PROGRAM MAIN
VAR
	//Matrix instances
	fbDispenseMatrix : FB_Matrix;
	fbInletMatrix : FB_Matrix;
	fbFillMatrix : FB_Matrix;

	//Instance of fbIO for IO updates
	fbIO : FB_IO;
	
	//Pressure Transducers
	aPT : ARRAY [1.. GVL_IO.cNumofPT] OF FB_PressureTransducer;
	
	//Devices interface
	Devices : ARRAY[1..GVL_IO.cNumofMatrices+GVL_IO.cNumofPT] OF I_Devices;
	
	//Initialising Boolean 
	bInitialise : BOOL := TRUE;
	
	idx : USINT;
	
	hr : HRESULT := S_PENDING;
END_VAR

//Run Initialise Method once on first cycle
IF bInitialise THEN
	hr := M_Initalize();
	RETURN;
END_IF

//Update IO
M_UpdateIO(PTTT:=aPT);

//Update From HMI
M_UpdateFromHMI();	

//Calling Cyclic
M_CyclicLogic();

//Update HMI
M_UpdateToHMI();

METHOD M_CyclicLogic
FOR idx := 1 TO GVL_IO.cNumofMatrices+GVL_IO.cNumofPT DO
    Devices[idx].M_CyclicLogic();
END_FOR
END_METHOD

METHOD PUBLIC M_Initalize : HRESULT
VAR
idx : INT;
// Config Parameter Struct 
stAnalogCfg : ST_AnalogPressureTemp;
hresult: ARRAY[1..GVL_IO.cNumofMatrices] OF HRESULT;
END_VAR

//Assign Devices into Interface array
Devices[1] := fbDispenseMatrix;
Devices[2] := fbInletMatrix;
Devices[3] := fbFillMatrix;
	
FOR idx := 1 TO GVL_IO.cNumofPT DO
    Devices[GVL_IO.cNumofMatrices + idx] := aPT[idx];
END_FOR
	
//Initialise the pressure sensors
FOR idx:=1 TO GVL_IO.cNumofPT DO
    aPT[idx].M_Init(sTag:=GVL_IO.sPTTags[idx]);
END_FOR

//Initialise matrices 
hresult[1] := fbInletMatrix.M_Init(nRows:=GVL_HMI.cInletRows,nCols:=GVL_HMI.cInletCols);
hresult[2] :=fbDispenseMatrix.M_Init(nRows:=GVL_HMI.cMaxRows,nCols:=GVL_HMI.cMaxCols);
hResult[3] := fbFillMatrix.M_Init(nRows:=GVL_HMI.cMaxRows,nCols:=GVL_HMI.cMaxCols);

//Logic to check if matrices fail to initialise
FOR idx:= 1 TO GVL_IO.cNumofMatrices DO
	IF hresult[idx] = E_FAIL THEN
		M_Initalize:= E_FAIL;
		RETURN;
	END_IF
END_FOR

//Initialised succesfully
bInitialise:=FALSE;
M_Initalize := S_OK;
END_METHOD

METHOD M_UpdateFromHMI
//Update each matrix using its update method
fbDispenseMAtrix.M_UpdateFromHMI(stHMI:=GVL_HMI.stDispHMI,
	                             nStartOfPath:=GVL_HMI.eDispStartOfPath,
								 nEndOfPath:=GVL_HMI.eDispEndOfPath);
								 
fbFillMatrix.M_UpdateFromHMI(stHMI:=GVL_HMI.stFillHMI,
	                             nStartOfPath:=GVL_HMI.eFillStartOfPath,
								 nEndOfPath:=GVL_HMI.eFillEndOfPath);
								 
fbInletMatrix.M_UpdateFromHMI(stHMI:=GVL_HMI.stInletHMI,
	                             nStartOfPath:=GVL_HMI.eInletStartOfPath,
								 nEndOfPath:=GVL_HMI.eInletEndOfPath);
END_METHOD

METHOD M_UpdateIO 
VAR_INPUT
	PTTT: REFERENCE TO ARRAY [1.. GVL_IO.cNumofPT] OF FB_PressureTransducer;
END_VAR
fbIO.DispenseMatrix:=fbDispenseMatrix;
fbIO.FillMatrix:=fbFillMatrix;
fbIO.InletMatrix:=fbInletMatrix;
fbIO(PTTT:=aPT);
END_METHOD

METHOD M_UpdateToHMI
VAR
	idx : INT;
END_VAR
fbDispenseMatrix.M_UpdateToHMI(stHMI:=GVL_HMI.stDispHMI);
fbFillMatrix.M_UpdateToHMI(stHMI:=GVL_HMI.stFillHMI);
fbInletMatrix.M_UpdateToHMI(stHMI:=GVL_HMI.stInletHMI);
FOR idx:=1 TO GVL_IO.cNumofPT DO
	aPT[idx].M_UpdateToHMI(PV=>GVL_HMI.aPV[idx],
		                   TV=>GVL_HMI.aTV[idx],
						   State=>GVL_HMI.aSensorErrors[idx]);
END_FOR
END_METHOD

END_PROGRAM

(* stored: Version 1.1.0.1
   POU MAIN: Id {606a3699-021a-464e-b575-9f2f01835131}, SpecialFunc None
   Folder Updates: Id {6a391c12-a86f-41a0-abbe-695c56b3d320}
   Method M_CyclicLogic: Id {d48a70cc-c9ea-409a-a41a-eae2b0a1f380}
   Method M_Initalize: Id {c8c10e44-8587-4199-9743-e05feaa06a39}
   Method M_UpdateFromHMI: Id {8779a328-bd71-463f-a457-6702a1e02170}
   Method M_UpdateIO: Id {b3dc1e8e-ddce-4750-a359-be425c8195a4}
   Method M_UpdateToHMI: Id {dc0c917a-29fb-4fe9-9454-5c7004a311f7} *)
